FUNCTION_BLOCK EL3174
VAR
	_io : EL3xx4_Data;
	{attribute addProperty Name "WcState"}
	_wcState : WcStateInputToggle;
	{attribute addProperty Name "Info data"}
	_infoData : InfoDataAds;
END_VAR

PROPERTY IO : REFERENCE TO EL3xx4_Data
GET
IO REF= _io;
END_GET
END_PROPERTY

PROPERTY WcState : REFERENCE TO WcStateInputToggle
GET
WcState REF= _wcState;
END_GET
END_PROPERTY

END_FUNCTION_BLOCK

(* stored: Version 1.1.0.1, ProductVersion 3.1.4024.9
   POU EL3174: Id {3019437b-a6fa-0aed-33ac-5774ba2c709f}, SpecialFunc None
   Property IO: Id {984646f1-b582-0c36-2f22-64ba1032f0fe}
   Get Get: Id {90ba4a6b-08b4-00bd-109a-2f1ad113f298}
   Property WcState: Id {4d3599ad-d21f-0399-171b-d3770fe7f396}
   Get Get: Id {fb1165cd-f27d-00db-02cc-a0979413c756} *)
